PROGRAM Inversores
VAR

(*=========================		INVERSORES		==========================*)	

	PassoMesaIndexAutomatico		: INT;
	PassoMesaIndexCiclo				: INT;
	PassoMesaIndexFwd				: INT;
	PassoMesaIndexBwd				: INT;
	PassoEsteiraSaidaAutomatico		: INT;
	PassoEsteiraSaidaFwd			: INT;
	PassoEsteiraSaidaBwd			: INT;

	TON_DelayParadaAuto				: TON;
	TON_DelayParadaCiclo			: TON;
	
	DelayParada						: TIME;
	
(*========================================================================*)

END_VAR

(*==============		SET Velocidade da Mesa Index		==============*)

FrequenciaMesaIndex := (INT_TO_REAL(IhmEscr_MesaIndex_Frequencia)/60)*(32767);
DelayParada	:= REAL_TO_TIME(IhmEscr_MesaIndex_DelayParada*1000);

(*=================		INVERSOR 1 - Mesa Index		======================*)

(*======================		Modo Automático		======================*)

//Condição de Bloqueio da Máquina de Estados - Mesa Index Automático
IF (Alarmes.AlarmeGrave
	//OR Alarmes.AlarmeMedio
	//OR Alarmes.AlarmeLeve
	OR NOT MaquinaLigada
	OR NOT MaquinaModoAuto
	OR NOT((ReguaPotenciometricaPosicao > ReguaPotenciometrica_Recuada_LI) AND (ReguaPotenciometricaPosicao < ReguaPotenciometrica_Recuada_LS))
	OR (NOT InSafety_CortinaLuz AND (PassoMesaIndexAutomatico > 13))
	) THEN
	PassoMesaIndexAutomatico := 1000;
	TON_DelayParadaAuto(IN:=FALSE);
	Flag_MesaIndex_Maquina := FALSE;
	LigarMesaIndexAutomatico := FALSE;	
END_IF

CASE PassoMesaIndexAutomatico OF
	
	//Passo 0 - Inicialização	
	0: PassoMesaIndexAutomatico := 10;
	
	//Passo 10 - Condição para Iniciar a Rotina Mesa Index (Sentido Normal - Automatico)
	10: IF  (Flag_Maquina_MesaIndex) THEN
			Flag_Maquina_MesaIndex := FALSE;
			PassoMesaIndexAutomatico := 11;
		END_IF

	//Passo 11 - Barreira Livre - Início do Processo
	11: IF  (InSafety_CortinaLuz) THEN
			PassoMesaIndexAutomatico := 12;
		END_IF
		
	//Passo 12 - Barreira Rompida - Posicionar Peça
	12: IF  (NOT InSafety_CortinaLuz) THEN
			PassoMesaIndexAutomatico := 13;
		END_IF
		
	//Passo 13 - Barreira Livre - Iniciar Movimentação da Mesa
	13: IF  (InSafety_CortinaLuz) THEN
			PassoMesaIndexAutomatico := 14;
		END_IF
		
	//Passo 14 - Movimentar Mesa Index
	14: LigarMesaIndexAutomatico := TRUE;
		
		Flag_Maquina_MesaIndex := FALSE;//Fora de posição para efeito de testes
	
		PassoMesaIndexAutomatico := 20;

	//Passo 20 - Aguardar Acionamento do Sensor de Posição 
	20: IF  InSensorIndutivo07 THEN
			PassoMesaIndexAutomatico := 30;	
		END_IF
	
	//Passo 30 - Aguardar Desacionamento do Sensor de Posição 
	30: IF  NOT InSensorIndutivo07 THEN
			PassoMesaIndexAutomatico := 40;	
		END_IF	

	//Passo 40 - Condição para Desligar Mesa Index - Delay de Parada
	40: TON_DelayParadaAuto(IN:=TRUE,PT:= DelayParada);
		IF (TON_DelayParadaAuto.Q) THEN
			TON_DelayParadaAuto(IN:=FALSE);
			LigarMesaIndexAutomatico := FALSE;
			PassoMesaIndexAutomatico := 50;
		END_IF
	
	//Passo 50 - Sinalização da Conclusão do Movimento
	50: Flag_MesaIndex_Maquina := TRUE;
		PassoMesaIndexAutomatico := 1000;
			
	//Passo 1000 - Finalização
	1000: PassoMesaIndexAutomatico := 0;
	
END_CASE

(*========================================================================*)

(*=========================		Modo Ciclo		==========================*)

//Condição de Bloqueio da Máquina de Estados - Mesa Index Ciclo
IF (Alarmes.AlarmeGrave 
	OR NOT MaquinaModoManual
	OR NOT InSafety_CortinaLuz
	) THEN
	PassoMesaIndexCiclo := 1000;
	TON_DelayParadaCiclo(IN:=FALSE);
	LigarMesaIndexCiclo := FALSE;
END_IF

CASE PassoMesaIndexCiclo OF
	
	//Passo 0 - Inicialização	
	0: PassoMesaIndexCiclo := 10;
	
	//Passo 10 - Condição para Ligar Mesa Index (Sentido Normal - Ciclo)
	10: IF  (IhmBt_MesaIndex_Ciclo) THEN
			PassoMesaIndexCiclo := 20;
		END_IF
		
	//Passo 20 - Aguardar o Botão Retorno do Botão
	20: IF  (NOT IhmBt_MesaIndex_Ciclo) THEN
			PassoMesaIndexCiclo := 30;
		END_IF
 
	//Passo 30 - Ligar Mesa Index
	30: LigarMesaIndexCiclo := TRUE;
		IF (InSensorIndutivo07) THEN
			PassoMesaIndexCiclo := 40;	
		END_IF
		
	//Passo 40 - Aguardar Desacionamento do Sensor de Posição 
	40:	IF (NOT InSensorIndutivo07) THEN
			PassoMesaIndexCiclo := 50;	
		END_IF

	//Passo 50 - Condição para Desligar Mesa Index 
	50: TON_DelayParadaCiclo(IN:=TRUE,PT:= DelayParada);
		IF (TON_DelayParadaCiclo.Q) THEN
			TON_DelayParadaCiclo(IN:=FALSE);
			LigarMesaIndexCiclo := FALSE;
			PassoMesaIndexCiclo := 1000;
		END_IF
			
	//Passo 1000 - Finalização
	1000: PassoMesaIndexCiclo := 0;
	
END_CASE

(*========================================================================*)

(*======================		Modo Manual		==========================*)

//Condição de Bloqueio da Máquina de Estados - Mesa Index FWD
IF (Alarmes.AlarmeGrave
	OR NOT MaquinaModoManual
	OR(NOT IhmBt_MesaIndex_LigarDesligar AND IhmBt_MesaIndex_Sentido)
	OR IhmBt_MesaIndex_Ciclo
	OR NOT InSafety_CortinaLuz
	) THEN
	PassoMesaIndexFwd := 1000;
	LigarMesaIndexFwd := FALSE;
	IhmBt_MesaIndex_LigarDesligar := FALSE;
END_IF

CASE PassoMesaIndexFwd OF
	
	//Passo 0 - Inicialização	
	0: PassoMesaIndexFwd := 10;
	
	//Passo 10 - Condição para Ligar Mesa Index (Sentido Normal - Forward)
	10: IF (NOT IhmBt_MesaIndex_Sentido AND IhmBt_MesaIndex_LigarDesligar) THEN
			LigarMesaIndexFwd := TRUE;
			PassoMesaIndexFwd := 20;
		END_IF

	//Passo 20 - Condição para Desligar Mesa Index 
	20: IF (NOT IhmBt_MesaIndex_LigarDesligar) THEN
			LigarMesaIndexFwd := FALSE;
			PassoMesaIndexFwd := 1000;	
		END_IF
	
	//Passo 1000 - Finalização
	1000: PassoMesaIndexFwd := 0;
	
END_CASE

//Condição de Bloqueio da Máquina de Estados - Mesa Index REV
IF (Alarmes.AlarmeGrave
	//OR NOT MaquinaModoManual
	//OR(NOT IhmBt_MesaIndex_LigarDesligar AND NOT IhmBt_MesaIndex_Sentido)
	OR IhmBt_MesaIndex_Ciclo
	) THEN
	PassoMesaIndexBwd := 1000;
	LigarMesaIndexBwd := FALSE;
	IhmBt_MesaIndex_LigarDesligar := FALSE;
END_IF

CASE PassoMesaIndexBwd OF
	
	//Passo 0 - Inicialização	
	0: PassoMesaIndexBwd := 10;
	
	//Passo 10 - Condição para Ligar Mesa Index (Sentido Reverso - Reverse)
	10: IF (IhmBt_MesaIndex_Sentido AND IhmBt_MesaIndex_LigarDesligar) THEN
			LigarMesaIndexBwd := TRUE;
			PassoMesaIndexBwd := 20;
		END_IF

	//Passo 20 - Condição para Desligar Mesa Index 
	20: IF (NOT IhmBt_MesaIndex_LigarDesligar) THEN
			LigarMesaIndexBwd := FALSE;
			PassoMesaIndexBwd := 1000;	
		END_IF
	
	//Passo 1000 - Finalização
	1000: PassoMesaIndexBwd := 0;
	
END_CASE

(*=============		SET Velocidade da Esteira de Saída		==============*)

FrequenciaEsteiraSaida := (INT_TO_REAL(IhmEscr_EsteiraSaida_Frequencia)/60)*(32767);

(*=============		INVERSOR 2 - Esteira de Saída		==================*)

(*======================		Modo Automático		======================*)



(*======================		Modo Manual		==========================*)

//Condição de Bloqueio da Máquina de Estados - Esteira de Saída FWD
IF (Alarmes.AlarmeGrave
	OR NOT MaquinaModoManual
	OR(NOT IhmBt_EsteiraSaida_LigarDesligar AND IhmBt_EsteiraSaida_Sentido)
	) THEN
	PassoEsteiraSaidaFwd := 1000;
	LigarEsteiraSaidaFwd := FALSE;
END_IF

CASE PassoEsteiraSaidaFwd OF
	
	//Passo 0 - Inicialização	
	0: PassoEsteiraSaidaFwd := 10;
	
	//Passo 10 - Condição para Ligar Esteira de Saída (Sentido Normal - Forward)
	10: IF (NOT IhmBt_EsteiraSaida_Sentido AND IhmBt_EsteiraSaida_LigarDesligar) THEN
			LigarEsteiraSaidaFwd := TRUE;
			PassoEsteiraSaidaFwd := 20;
		END_IF

	//Passo 20 - Condição para Desligar Esteira de Saída 
	20: IF (NOT IhmBt_EsteiraSaida_LigarDesligar) THEN
			LigarEsteiraSaidaFwd := FALSE;
			PassoEsteiraSaidaFwd := 1000;	
		END_IF
	
	//Passo 1000 - Finalização
	1000: PassoEsteiraSaidaFwd := 0;
	
END_CASE

//Condição de Bloqueio da Máquina de Estados - Esteira de Saída REV
IF (Alarmes.AlarmeGrave
	//OR NOT MaquinaModoManual
	OR(NOT IhmBt_EsteiraSaida_LigarDesligar AND NOT IhmBt_EsteiraSaida_Sentido)
	) THEN
	PassoEsteiraSaidaBwd := 1000;
	LigarEsteiraSaidaBwd := FALSE;		
END_IF

CASE PassoEsteiraSaidaBwd OF
	
	//Passo 0 - Inicialização	
	0: PassoEsteiraSaidaBwd := 10;
	
	//Passo 10 - Condição para Ligar Mesa Index (Sentido Reverso - Reverse)
	10: IF (IhmBt_EsteiraSaida_Sentido AND IhmBt_EsteiraSaida_LigarDesligar) THEN
			LigarEsteiraSaidaBwd := TRUE;
			PassoEsteiraSaidaBwd := 20;
		END_IF

	//Passo 20 - Condição para Desligar Mesa Index 
	20: IF (NOT IhmBt_EsteiraSaida_LigarDesligar) THEN
			LigarEsteiraSaidaBwd := FALSE;
			PassoEsteiraSaidaBwd := 1000;	
		END_IF
	
	//Passo 1000 - Finalização
	1000: PassoEsteiraSaidaBwd := 0;
	
END_CASE

(*========================================================================*)

(*=====================		INVERSORES	- SAÍDAS	======================*)	

//Inversor 1 - Mesa Index
IF (LigarMesaIndexFwd OR LigarMesaIndexCiclo OR LigarMesaIndexAutomatico) THEN
	OutSentidoGiroMesaIndex := FALSE;
	OutLigarMesaIndex := TRUE;
ELSIF (LigarMesaIndexBwd) THEN
	OutSentidoGiroMesaIndex := TRUE;
	OutLigarMesaIndex := TRUE;
ELSE
	OutSentidoGiroMesaIndex := FALSE;
	OutLigarMesaIndex := FALSE;
END_IF

//Inversor 2 - Esteira de Saída
IF (LigarEsteiraSaidaFwd) THEN
	OutSentidoGiroEsteiraSaida := FALSE;
	OutLigarEsteiraSaida := TRUE;
ELSIF (LigarEsteiraSaidaBwd) THEN
	OutSentidoGiroEsteiraSaida := TRUE;
	OutLigarEsteiraSaida := TRUE;
ELSE
	OutSentidoGiroEsteiraSaida := FALSE;
	OutLigarEsteiraSaida := FALSE;
END_IF

(*========================================================================*)

END_PROGRAM

(* stored: Version 1.1.0.1, ProductVersion 3.1.4024.11
   POU Inversores: Id {9cc97f29-a3ae-4037-90a4-ce9c90bf4f32}, SpecialFunc None *)
